{attribute 'qualified_only' := ''}
{attribute 'strict' := ''}
TYPE RudongPump_ERROR_1 :
(
	No_ERROR := 0,
	/// E-Gripper Parameter fault   程序配置参数有问题 
	FLT_PARA := 1,
	/// E-Gripper not ready 旋转有通信报警
	FLT_CONNECT := 2,
	/// E-Gripper read/write command while not ready 预留
	FLT_RDYCMD := 3,
	/// 配置参数错误 
	FLT_CONFIGURE_PARA := 4,
	/// 流量时间配置错误 
	FLT_FLUVOLUM_TIME_PARA := 5,
	/// E-Gripper release  execute Timeout 
	FLT_PUSH_TIMEOUT := 10,
	/// E-Gripper org  execute Timeout 
	FLT_PULL_TIMEOUT := 11,
	/// E-Gripper org command execute Timeout 
	FLT_STOP_TIMEOUT := 12,
	/// E-Gripper org command execute Timeout 
	FLT_FULLSPEEDSTOP_TIMEOUT := 13,
	/// E-Gripper org command execute Timeout 
	FLT_FULLSPEEDSTART_TIMEOUT := 14,
	/// E-Gripper release command execute Timeout 
	FLT_CMD_TIMEOUT := 15,
	/// E-Gripper release command execute Timeout 
	FLT_RUN_FALL := 16,
	/// E-Gripper org  execute Timeout 
	FLT_PumpCal_TIMEOUT := 17,
	/// E-Gripper org  execute Timeout 
	FLT_PumpCal_OverFlow := 18,
	/// Modbus 
	FLT_Mobdus := 19
);
END_TYPE

(* stored: Version 1.1.0.1, ProductVersion 3.1.4024.9
   DUT RudongPump_ERROR_1: Id {151a99aa-6537-4039-bf7b-e8aa6ba00d39} *)
